FUNCTION Convert_ULINT_TO_DATE : Hresult
VAR_INPUT
	in : ULINT;
	out : REFERENCE TO DATE;
END_VAR
VAR
	converted : DATE;
END_VAR

converted := ULINT_TO_DATE(in);

IF (DATE_TO_ULINT(converted) <> in) THEN
	Convert_ULINT_TO_DATE := INCOMPATIBLE;
	RETURN;
END_IF

out := converted;

END_FUNCTION

(* stored: Version 1.1.0.1, ProductVersion 3.1.4024.12
   POU Convert_ULINT_TO_DATE: Id {06c0b158-05eb-46c5-977e-54cf690af4b6}, SpecialFunc None *)
